Yaskawa INFORM job: B-9-08279-80-90-L.JBI

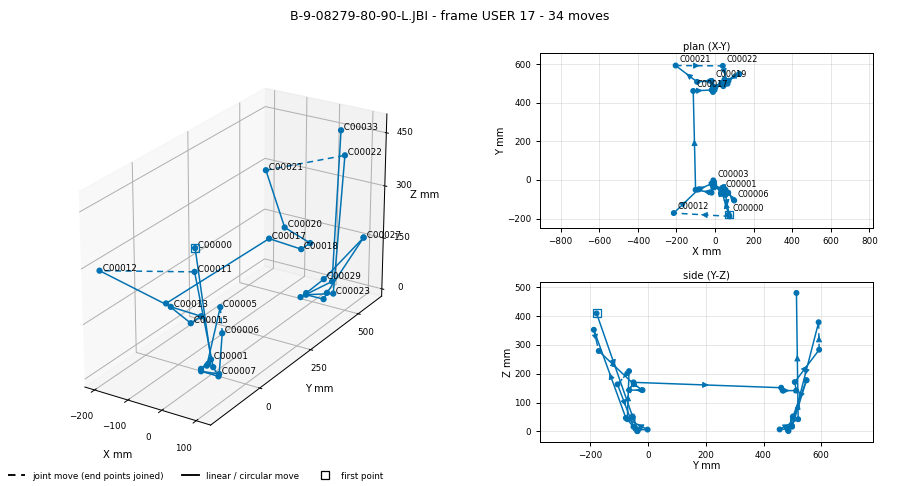
[picture p0: tool path of B-9-08279-80-90-L.JBI in frame USER 17, 34 of 34 moves have a stored position in this frame; points joined in program order, loops and branches not executed]
/JOB
//NAME B-9-08279-80-90-L
///FOLDERNAME PART_420-08279-80
//POS
///NPOS 34,0,34,0,0,0
///USER 17
///TOOL 4
///POSTYPE USER
///RECTAN
///RCONF 1,0,0,0,0,0,0,0,0,0,0,0,0,0,0,0,0,0,0,0,0,0,0,0
C00000=70.970,-178.868,409.213,-165.0000,45.0000,0.0000
C00001=33.224,-54.308,52.156,-165.0000,45.0000,0.0000
C00002=-8.772,-35.324,6.270,178.9998,57.8139,-39.3487
C00003=-8.695,-1.943,6.305,178.9069,57.7755,-44.4758
C00004=32.283,-72.150,42.455,-165.0000,45.0000,0.0000
C00005=68.685,-66.272,209.042,-165.0000,45.0000,0.0000
C00006=99.538,-106.298,163.160,-166.3780,45.3490,-50.4350
C00007=54.868,-50.966,16.241,133.5610,7.6410,-152.0390
C00008=-7.079,-37.865,1.257,126.4294,11.4889,-151.1171
C00009=44.023,-37.162,0.732,126.4299,11.4905,-151.1166
C00010=54.426,-77.432,46.656,126.4293,11.4917,-151.1175
C00011=75.120,-188.373,352.355,175.5546,51.6267,-23.6686
C00012=-213.482,-171.326,278.744,154.4200,34.7310,45.4810
C00013=-87.212,-49.799,163.694,107.6090,9.3560,77.2190
C00014=-17.742,-19.511,143.212,104.0909,8.5652,76.6643
C00015=-17.848,-65.814,143.146,104.0918,8.5656,76.6647
C00016=-100.598,-50.810,170.079,107.6090,9.3560,77.2190
C00017=-112.794,461.129,151.518,107.5190,-7.4490,103.3910
C00018=-16.732,466.487,141.430,98.4465,-5.2396,104.4229
C00019=-16.623,513.278,141.483,98.4467,-5.2394,104.4226
C00020=-92.930,508.215,171.083,107.5190,-7.4490,103.3910
C00021=-203.967,592.873,283.205,107.5190,-7.4490,103.3910
C00022=40.454,590.981,378.479,-169.5230,46.0050,83.6620
C00023=64.926,498.805,18.936,-133.5620,7.6410,152.0390
C00024=-11.200,486.062,1.710,-133.5656,7.6431,152.0306
C00025=42.872,485.949,2.186,-133.5658,7.6407,152.0341
C00026=45.609,498.918,16.234,-144.8388,26.9003,148.6583
C00027=125.350,548.745,177.334,165.0001,45.0004,0.0014
C00028=125.357,548.743,177.335,165.0000,45.0000,0.0000
C00029=33.224,502.241,52.156,165.0000,45.0000,0.0000
C00030=-9.168,483.281,8.252,165.0891,51.2742,6.9893
C00031=-10.607,455.830,6.834,165.1632,51.2621,15.5387
C00032=48.694,520.054,42.252,165.0010,44.9996,-0.0009
C00033=70.181,514.089,480.075,165.0008,44.9999,-0.0009
///POSTYPE ANGLE
///ANGLE
EC00000=90.0000
EC00001=90.0000
///TOOL 0
EC00002=90.0000
EC00003=90.0000
///TOOL 4
EC00004=90.0000
EC00005=90.0000
EC00006=105.0000
EC00007=105.0000
///TOOL 0
EC00008=105.0000
EC00009=105.0000
EC00010=105.0000
EC00011=105.0000
///TOOL 4
EC00012=135.0000
EC00013=135.0000
///TOOL 0
EC00014=135.0000
EC00015=135.0000
///TOOL 4
EC00016=135.0000
EC00017=135.0000
///TOOL 0
EC00018=135.0000
EC00019=135.0000
///TOOL 4
EC00020=135.0000
EC00021=135.0000
EC00022=105.0000
EC00023=105.0000
///TOOL 0
EC00024=105.0000
EC00025=105.0000
EC00026=105.0000
EC00027=90.0000
///TOOL 4
EC00028=90.0000
EC00029=90.0000
///TOOL 0
EC00030=90.0000
EC00031=90.0000
EC00032=90.0000
EC00033=90.0000
//INST
///DATE 2021/10/29 11:36
///ATTR SC,RW,RJ
////FRAME USER 17
///GROUP1 RB1
///GROUP2 ST3
NOP
'Path Start: PP1_1
MOVJ C00000 VJ=100.00  +MOVJ EC00000
SMOVL C00001 V=1250.0  +MOVJ EC00001
SMOVL C00002 V=1250.0  +MOVJ EC00002
ARCON ASF#(951)
SMOVL C00003 V=8.5  +MOVJ EC00003
ARCOF AEF#(951)
SMOVL C00004 V=1250.0  +MOVJ EC00004
SMOVL C00005 V=1250.0  +MOVJ EC00005
'Path End
'Path Start: PP48
MOVJ C00006 VJ=100.00  +MOVJ EC00006
SMOVL C00007 V=1250.0  +MOVJ EC00007
SMOVL C00008 V=300.0  +MOVJ EC00008
ARCON ASF#(953)
SMOVL C00009 V=15.7  +MOVJ EC00009
ARCOF AEF#(953)
SMOVL C00010 V=1250.0  +MOVJ EC00010
SMOVL C00011 V=1250.0  +MOVJ EC00011
'Path End
'Path Start: PP47
MOVJ C00012 VJ=100.00  +MOVJ EC00012
SMOVL C00013 V=1250.0  +MOVJ EC00013
SMOVL C00014 V=300.0  +MOVJ EC00014
ARCON ASF#(953)
SMOVL C00015 V=12.7  +MOVJ EC00015
ARCOF AEF#(953)
SMOVL C00016 V=1250.0  +MOVJ EC00016
'Path End
'Path Start: PP42
SMOVL C00017 V=1250.0  +MOVJ EC00017
SMOVL C00018 V=300.0  +MOVJ EC00018
ARCON ASF#(953)
SMOVL C00019 V=12.7  +MOVJ EC00019
ARCOF AEF#(953)
SMOVL C00020 V=1250.0  +MOVJ EC00020
SMOVL C00021 V=1250.0  +MOVJ EC00021
'Path End
'Path Start: PP41
MOVJ C00022 VJ=100.00  +MOVJ EC00022
SMOVL C00023 V=1250.0  +MOVJ EC00023
SMOVL C00024 V=300.0  +MOVJ EC00024
ARCON ASF#(953)
SMOVL C00025 V=15.7  +MOVJ EC00025
ARCOF AEF#(953)
SMOVL C00026 V=1250.0  +MOVJ EC00026
SMOVL C00027 V=1250.0  +MOVJ EC00027
'Path End
'Path Start: PP1
MOVJ C00028 VJ=100.00  +MOVJ EC00028
SMOVL C00029 V=1250.0  +MOVJ EC00029
SMOVL C00030 V=1250.0  +MOVJ EC00030
ARCON ASF#(951)
SMOVL C00031 V=8.5  +MOVJ EC00031
ARCOF AEF#(951)
SMOVL C00032 V=1250.0  +MOVJ EC00032
SMOVL C00033 V=1250.0  +MOVJ EC00033
INC I005
'Path End
END
